FUNCTION Value : I_BoolValue
VAR_INPUT
	boolean : REFERENCE TO BOOL;
END_VAR
VAR
	p : POINTER TO FB_BoolBindingReadOnly;
END_VAR

p := __NEW(FB_BoolBindingReadOnly);

p^.Bind(boolean);

Value := p^;

END_FUNCTION

(* stored: Version 1.1.0.1
   POU Value: Id {90e98975-5217-4b6e-97cc-fa4c6cc2a31b}, SpecialFunc None *)
